// TIA Portal V16 export
// export: Created 2021-11-12T13:31:57.5725382Z, ExportSetting WithDefaults, DisplayName Totally Integrated Automation Portal, DisplayVersion V16 Update 3, DisplayName TIA Portal Version Control Interface, DisplayVersion V16 Update 2, DisplayName TIA Portal Openness, DisplayVersion V16 Update 3, DisplayName SINAMICS Startdrive Advanced, DisplayVersion V16 Update 5, DisplayName SINAMICS Startdrive G130, G150, S120, S150, SINAMICS MV, S210, DisplayVersion V16 Update 5, DisplayName SINAMICS Startdrive G110M, G120, G120C, G120D, G120P, G115D, DisplayVersion V16 Update 5, DisplayName STEP 7 Professional, DisplayVersion V16 Update 3, DisplayName STEP 7 Safety, DisplayVersion V16, DisplayName WinCC UA Professional, DisplayVersion V16 Update 3
DATA_BLOCK "IDB_Cab_000+UC20_DB"   // DB215
VERSION : 0.1
// stored: AutoNumber true, DBAccessibleFromOPCUA true, InstanceOfName Cab_000+UC20, InstanceOfType FB
"Cab_000+UC20"
   // VAR
   //    "SF_000UC20-FB21_14_Alarm" { S7_SetPoint := 'True'} : "STD_DI_Mon";
   //    "SF_000UC20-FC21_14_Alarm" { S7_SetPoint := 'True'} : "STD_DI_Mon";
   //    "SF_000UC20-EC01_3_Alarm" { S7_SetPoint := 'True'} : "STD_DI_Mon";
   //    "SF_000UC20-FC01_14_Alarm" { S7_SetPoint := 'True'} : "STD_DI_Mon";
   //    "SF_000UC20-TB01_14_Alarm" { S7_SetPoint := 'True'} : "STD_DI_Mon";
   //    "SF_000UC20-FC30_14_Alarm" { S7_SetPoint := 'True'} : "STD_DI_Mon";
   //    "SF_000UC20-FC30_24_Alarm" { S7_SetPoint := 'True'} : "STD_DI_Mon";
   //    "SF_000UC20-FC50_14_Alarm" { S7_SetPoint := 'True'} : "STD_DI_Mon";
   //    "SF_000UC20-FC50_24_Alarm" { S7_SetPoint := 'True'} : "STD_DI_Mon";
   // END_VAR
BEGIN
END_DATA_BLOCK
